{attribute addProperty BoxType "EL2521-0000-1019"}
{attribute addProperty Id "StatusAT %I*Status_D2AF8223162"}
{attribute addProperty CRC "884081489"}
{attribute addProperty SizeInBites "16"}
{attribute addProperty SizeInBytes "2"}
TYPE PTO_Status_34B20351 :
STRUCT
	{attribute addProperty Name "Status"}
	Status AT %I* : Status_D2AF8223;
END_STRUCT
END_TYPE

(* stored: Version 1.2.0.0, ProductVersion 3.1.4024.9
   DUT PTO_Status_34B20351: Id {51a91da6-29bc-4237-a097-1222da26b137} *)
